// TIA Portal V20 export
DATA_BLOCK "instFB_Init"   // DB22
VERSION : 1.1
// Instance DB for FB_Init (Phase 3, 2026-05-21). Homing block - LKinCtrl_MC_GroupHome on ScaraArm3D, runs in OB30. DB number may be auto-assigned by TIA on import.
// stored: InstanceOfName FB_Init, InstanceOfType FB
"FB_Init"
   // VAR
   //    instGroupHome { S7_SetPoint := 'True'} : "LKinCtrl_MC_GroupHome";
   // END_VAR
BEGIN
END_DATA_BLOCK
